FUNCTION_BLOCK E_DEMUX_5 (* Event demultiplexer (generic FB) *)
  (* Standard: 61499-1 Annex A; Description: Copyright (c) 2025 Martin Erich Jobst This program and the accompanying materials are made available under the terms of the Eclipse Public License 2.0 which is available at https://www.eclipse.org/legal/epl-2.0/ SPDX-License-Identifier: EPL-2.0 *)
  (* Version 3.0, 2025-08-25, Martin Erich Jobst, initial API and implementation and/or initial documentation *)
  PACKAGE iec61499::events;
  {SET_ATTRIBUTE(eclipse4diac::core::GenericClassName, 'GEN_E_DEMUX')}
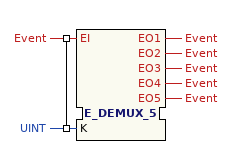
  EVENT_INPUT
    EI WITH K; (* Event to demultiplex *)
  END_EVENT
  EVENT_OUTPUT
    EO1; (* Output, demultiplexed from EI when K=0 *)
    EO2; (* Output, demultiplexed from EI when K=1 *)
    EO3; (* Output, demultiplexed from EI when K=2 *)
    EO4; (* Output, demultiplexed from EI when K=3 *)
    EO5; (* Output, demultiplexed from EI when K=4 *)
  END_EVENT
  VAR_INPUT
    K : UINT; (* Event index *)
  END_VAR
END_FUNCTION_BLOCK
